(* CoDeSys 2.3 export: GETEEP_INDEX.EXP *)

(* POU 05_Basic_Calc/eeprom_operations/getEEP_Index, ST *)
(* Функция получает номер ячейки относительно начала текущей страницы *)
FUNCTION getEEP_Index : INT
VAR_INPUT
	EEP_num					: INT;
END_VAR
VAR
	EEP_ELEMENT_OF_PAGE	: INT		:= 256;
END_VAR
getEEP_Index := EEP_num - (EEP_num / EEP_ELEMENT_OF_PAGE) * EEP_ELEMENT_OF_PAGE;
END_FUNCTION
